INTERFACE IStation

PROPERTY Busy : BOOL
GET
END_GET
END_PROPERTY

METHOD Execute : PVOID
VAR_INPUT
END_VAR
END_METHOD

PROPERTY Faulted : BOOL
GET
END_GET
END_PROPERTY

PROPERTY Ready : BOOL
GET
END_GET
END_PROPERTY

END_INTERFACE

(* stored: Version 1.1.0.1, ProductVersion 3.1.4024.12
   Itf IStation: Id {45cff2cc-58be-4c22-9fd9-11924f5790cb}
   Property Busy: Id {4fc5c0e7-13cf-4567-b2f5-677d7776b18e}
   Get Get: Id {04d7b57e-39b6-4240-ad95-769311436a15}
   Method Execute: Id {671ded2a-ae12-4b2a-bae9-8a08b12af770}
   Property Faulted: Id {7e549cf9-6633-4763-baf1-7c47845ee9f3}
   Get Get: Id {ed49b174-4b58-4ed6-9fd4-695014c6d0a1}
   Property Ready: Id {333f4836-c265-40d2-9ceb-b26b41d02803}
   Get Get: Id {bb6439fd-c1c5-4364-83ad-da8044e7442a} *)
